TYPE ST_ItemOUT3 :
STRUCT
	Identity		:ST_IdentityOUT3;
	ItemState		:STRING;
	RejectReason	:ST_RejectReasonOUT3;
	logs			:ST_logsOUT3;
	NoRead			:STRING;
	Content			:ST_ContentOUT3;
END_STRUCT
END_TYPE

(* stored: Version 1.1.0.1, ProductVersion 3.1.4024.13
   DUT ST_ItemOUT3: Id {3558badb-94e9-4d57-8da9-c3187af9548d} *)
